FUNCTION_BLOCK FB_PathUtilities IMPLEMENTS I_Path
VAR_INPUT
END_VAR
VAR_OUTPUT
END_VAR
VAR
	_pathGenerator	: FB_PathGenerator;
END_VAR

(* Checks if path exists, return TRUE when done and the result is returned in `result` output var.*)
METHOD Exists : BOOL
VAR_INPUT
	path	: Tc2_System.T_MaxString;
END_VAR
VAR_OUTPUT
	result	: BOOL;
END_VAR
END_METHOD

(* Generates the file path based on the location, file name and extension*)
METHOD Generate : I_PathGenerator
Generate := _pathGenerator;
END_METHOD

END_FUNCTION_BLOCK

(* stored: Version 1.1.0.1, ProductVersion 3.1.4024.14
   POU FB_PathUtilities: Id {aa4bc240-593b-0fc8-096f-eb4a070d9a09}, SpecialFunc None
   Method Exists: Id {91811280-46ee-03e8-22db-c845ddec0ad1}
   Method Generate: Id {57891d39-aafb-055c-337c-0e7884702c01} *)
